TYPE ST_JoystickScaling :
STRUCT
END_STRUCT
END_TYPE

(* stored: Version 1.1.0.1, ProductVersion 3.1.4024.12
   DUT ST_JoystickScaling: Id {8206ad67-42d5-45b3-a5f6-c9d08a2d3900} *)
